Staubli VAL3: onEdit.pgx

public program onEdit(string& x_sItem[] (dimensions=1))
  local num l_nResult
begin
  //
  // go to the view instruction page
  //
  if size(x_sItem)>1
    call load(x_sItem,l_nResult)
    // give it back
    x_sItem[1]=x_sItem
    x_sItem="Disk://instruction/PROG/page_viewInstr"
  endIf
end
